// TIA Portal V20 export
TYPE "UDT_OPC_Maintenance"
   STRUCT
      Elapsed : Real;   // Temps de fonctionnement actuel (en unité de temps)
      Id : Int;   // ID de la tache
      Period : Int;   // Durée maximale avant maintenance
      Reset : Bool;   // Reset Temps de fonctionnement actuel
      WarningThreshold : Int;   // Seuil d'avertissement en % (par défaut 80%)
   END_STRUCT;
END_TYPE
